VAR_GLOBAL CONSTANT
    TcUnit_ResultExportXmlPath : T_MaxString :=
        'C:\TwinCAT\3.1\Boot\Plc\TcUnitResults.xml';
END_VAR

(* stored: Version 1.1.0.1
   GVL GVL_TcUnit: Id {411aa615-69d5-432a-ab63-42412d812dc8} *)
